(* IEC 61131-3 sources: Industry-PLC-LLM/data/PLCBEAD_repo/PLCBEAD_PLCEmbed-main/PLC-BEAD/Source/GEB/CTANH, 1 file *)

(* ---- CTANH.ST ---- *)
TYPE oscat_complex :
  STRUCT
	re : REAL;
	im : REAL;
  END_STRUCT;
END_TYPE

FUNCTION COSH:REAL
	VAR_INPUT
		X :	REAL;
	END_VAR

	VAR
		T :	REAL;
	END_VAR

	T := EXP(X);
	COSH := (1.0 / T + T) * 0.5;
END_FUNCTION

FUNCTION SINH:REAL
	VAR_INPUT
		X :	REAL;
	END_VAR

	IF ABS(X) < 2.0E-3 THEN
		SINH := X;
	ELSE
		SINH := (EXP(X) - EXP(-X)) * 0.5;
	END_IF;
END_FUNCTION

FUNCTION_BLOCK CTANH_Block
	VAR_INPUT
		X :	oscat_complex;
	END_VAR

	VAR_OUTPUT
		CTANH :	oscat_complex;
	END_VAR

	VAR
		xi2 :	REAL;
		xR2 :	REAL;
		temp :	REAL;
	END_VAR

	xi2 := 2.0 * X.im;
	xR2 := 2.0 * X.re;
	temp := 1.0 /(COSH(xR2) + COS(xi2));
	CTANH.re := temp * SINH(xR2);
	CTANH.im := temp * SIN(xi2);

END_FUNCTION_BLOCK

PROGRAM program0
  VAR
    LocalVar0 : oscat_complex;
	LocalOUT  : oscat_complex;
	func_block : CTANH_Block;
  END_VAR
	func_block.X  := LocalVar0;
	func_block();
	LocalOUT := func_block.CTANH;
END_PROGRAM
